Staubli VAL3: remMovJointAxis.pgx

program remMovJointAxis(string& sArgs[] (dimensions=1), string& sReturn[] (dimensions=1))
  local bool bOk
  local joint jDest
  local num nIndex
  local num nVal
  local point pDest
  local string sAxis
  local string sVal
begin
  //Move just one joint
  //Arguments are "j pos" where j is J1, J2, J3, J4, J5, or J6 and pos is the goal
  //
  logMsg("call remMovJointAxis")
  nIndex=find(sArgs," ")
  sAxis=left(sArgs,nIndex)
  sVal=delete(sArgs,nIndex+1,0)
  toNum(sVal,nVal,bOk)
  if bOk
    jDest=herej()
    switch sAxis
      case "J1"
        jDest.j1=nVal
      break
      case "J2"
        jDest.j2=nVal
      break
      case "J3"
        jDest.j3=nVal
      break
      case "J4"
        jDest.j4=nVal
      break
      case "J5"
        jDest.j5=nVal
      break
      case "J6"
        jDest.j6=nVal
      break
      default
        call remErrInvalid("MOVJOINTAXIS",sAxis,sReturn)
        return
      break
    endSwitch
    if nIPNumber==0
      pDest=jointToPoint(tSensorTool,fIP1,jDest)
    else
      pDest=jointToPoint(tSensorTool,fIP2,jDest)
    endIf
    call remMovBase(pDest,sReturn)
  else
    call remErrNum("MOVJOINTAXIS",sVal,sReturn)
  endIf
end
